# EPICS autosave request: tomoScanApp/Db/tomoScan_PCO_settings.req
# Database for EPICS PVS for tomoScan using the EPICS motor record position compare output (PCO) support

################
# PCO Prefix
################
$(P)$(R)PCOPVPrefix
